{attribute 'linkalways'} 
{attribute 'no_explicit_call' := 'This FB is a CLASS and must be accessed using methods or properties'}
{attribute 'enable_dynamic_creation'}
FUNCTION_BLOCK MoveAbsoluteCommand EXTENDS Mc2MotionCommand
VAR
	fb : Tc2_Mc2.Mc_MoveAbsolute;
END_VAR

{attribute 'monitoring' := 'call'}
PROPERTY PUBLIC Active : BOOL
GET // PUBLIC
Active := fb.Active;
END_GET
END_PROPERTY

METHOD PUBLIC CyclicCall
SUPER^.CyclicCall();
fb(Axis := axis_ref);
END_METHOD

(*FB_Init is always available implicitly and it is used primarily for initialization.
The return value is not evaluated. For a specific influence, you can also declare the
methods explicitly and provide additional code there with the standard initialization
code. You can evaluate the return value.*)
METHOD FB_Init : BOOL
VAR_INPUT
	(* TRUE: the retain variables are initialized (reset warm / reset cold)*)
	bInitRetains : BOOL;
	(* TRUE: the instance will be copied to the copy code afterward (online change)*)
	bInCopyCode	: BOOL;
	axis : Axis;
	position : LREAL;
	velocity : LREAL;
	acceleration : LREAL := 0;
	deceleration : LREAL := 0;
	jerk : LREAL := 0;
	buffer_mode	: MotionBufferMode := MotionBufferMode.Aborting;
END_VAR
fb.Position := position;
fb.Velocity := velocity;
fb.Acceleration := acceleration;
fb.Deceleration := deceleration;
fb.Jerk := jerk;
fb.BufferMode := Mc2BufferModeConvertTo(buffer_mode);
END_METHOD

METHOD PROTECTED OnExecuting
VAR_INPUT
	state_control : AsyncCommandStateControl;
END_VAR
fb.Execute := TRUE;

IF fb.Done THEN
	fb.Execute := FALSE;
	state_control.Next();
END_IF

IF fb.CommandAborted THEN
	fb.Execute := FALSE;
	Abort();
END_IF

IF fb.Error THEN
	fb.Execute := FALSE;
	state_control.Error(fb.ErrorId);
END_IF
END_METHOD

END_FUNCTION_BLOCK

(* stored: Version 1.1.0.1
   POU MoveAbsoluteCommand: Id {e57e34b4-d39b-0329-15f2-c57e5828e3c8}, SpecialFunc None
   Property Active: Id {908a3ab5-e875-0625-030d-94f19ded8287}
   Get Get: Id {70fac97a-a517-04c7-22c4-42963c727b03}
   Method CyclicCall: Id {6dc2c71b-4e7d-0f13-072c-d64182173c58}
   Method FB_Init: Id {16cf053a-bc75-0eca-15e7-40da13d01a96}
   Method OnExecuting: Id {832add53-d405-0667-1b44-f13e26cc9567} *)
